PROGRAM PMPS
VAR
	fbArbiterIO : FB_SubSysToArbiter_IO;
END_VAR

fbArbiterIO(Arbiter := GVL_PMPS.g_fbArbiter1, fbFFHWO := GVL_PMPS.g_FastFaultOutput1);

END_PROGRAM

(* stored: Version 1.1.0.1, ProductVersion 3.1.4022.18
   POU PMPS: Id {3b7307dd-d4f5-405e-8e38-9780f4bf414e}, SpecialFunc None *)
